// TIA Portal V20 export
TYPE "ST_Motor"
   STRUCT
      Current : Real;
      State : Struct
         Run : Bool;
      END_STRUCT;
   END_STRUCT;
END_TYPE
